{attribute 'pack_mode' := '2'}
TYPE ST_DATA_CTRL :
STRUCT
  Cmd       : E_DATA_CTRL;
END_STRUCT
END_TYPE

(* stored: Version 1.1.0.1, ProductVersion 3.1.4026.20
   DUT ST_DATA_CTRL: Id {eaef2ff0-5a1c-4f88-8f58-2c2d2de8b75b} *)
